{attribute 'Tc2GvlVarNames'}
{attribute 'strict'}
TYPE e_ProgrammiMovimentoZ :
(
	
	Z_PosDiRiposo						:= 0,
	Z_PosFuoriIngombroRiposo 			:= 6,

	Z_PosStartLentaPrelievoFalda		:= 51,
	Z_PosPrelievoInLentaFalda 			:= 52,
	Z_PosAttesaCadutaFalda				:= 53,
	Z_PosFuoriIngombroFalda 			:= 54,
	Z_PosStartLentaDepositoSuCatasta	:= 55,
	Z_PosDepositoInLentaSuCatasta		:= 56,
	Z_PosStartLentaDepositoFalda		:= 57,
	Z_PosDepositoInLentaFalda			:= 58,

	Z_PosStartLentaPrelievoLastra 		:= 101,
	Z_PosPrelievoInLentaLastra 			:= 102,
	Z_PosDistaccoLastraInLentaLastra	:= 103,
	Z_PosStartLentaDepositoLastra 		:= 104,
	Z_PosDepositoInLentaLastra			:= 105,
	Z_PosFuoriIngombroVuotoLastra		:= 106,
	
	Z_PosFuoriIngombroCaricoLastra		:= 126,
	Z_PosPostScarico					:= 127
);
END_TYPE

(* stored: Version 1.1.0.1, ProductVersion 3.1.4024.11
   EnumerationTextList e_ProgrammiMovimentoZ: Id {9a655f4b-0810-43bf-91f4-d68484a40e94} *)
